{attribute 'enable_dynamic_creation'}
FUNCTION_BLOCK LineList EXTENDS CNM_AbstractObject.Object IMPLEMENTS ILineList
VAR
	list : CNM_Collections.ArrayList(1000);
END_VAR

(*

short summary
=================
This methode adds the given CNM_AbstractObject.IObject to the end of the list.
Example: 
Given a list that looks like this: (Head->) A B C (<- End),
calling append(D) on this list will place the D at the and,
making it the new End: (Head->) A B C D(<- End)

.. <legal notes>

legal notes
=================
| SPDX-FileCopyrightText: © 2022 ekvip automation GmbH <info@ekvip.de>
| SPDX-License-Identifier: Apache-2.0
| For details check: Apache-2.0_

.. _Apache-2.0: https://www.apache.org/licenses/LICENSE-2.0

.. </legal notes>

parameters
=================

*)
METHOD append : CNM_ReturnTypes.SingleExecutionResult
VAR_INPUT
	(*The object to be appended*)
	line	: ILine;
END_VAR
append := THIS^.list.append(object := line);
END_METHOD

(*

short summary
=================
This methode adds all elements of the given collection to the end of this list.
Example:
For the list1: A B C and list2: D E F will be after list1.appendCollection(list2):
A B C D E F. Notice the elements are still in the same order they where befor on each subsection.

.. <legal notes>

legal notes
=================
| SPDX-FileCopyrightText: © 2022 ekvip automation GmbH <info@ekvip.de>
| SPDX-License-Identifier: Apache-2.0
| For details check: Apache-2.0_

.. _Apache-2.0: https://www.apache.org/licenses/LICENSE-2.0

.. </legal notes>

parameters
=================

*)
METHOD appendCollection : CNM_ReturnTypes.SingleExecutionResult
VAR_INPUT
	(*The collection to be appended*)
	collectionToAppend	: CNM_CollectionInterfaces.ICollection;
END_VAR
appendCollection := THIS^.list.appendCollection(collectionToAppend);
END_METHOD

PROPERTY className : ClassName
GET
className := 'LineList';
END_GET
END_PROPERTY

(*

short summary
=================
This methode clears/deletes all clearable data from this object.
Example:
A list: 1 2 3 after list.clear() will have no remaining items, isEmpty = true.

.. <legal notes>

legal notes
=================
| SPDX-FileCopyrightText: © 2022 ekvip automation GmbH <info@ekvip.de>
| SPDX-License-Identifier: Apache-2.0
| For details check: Apache-2.0_

.. _Apache-2.0: https://www.apache.org/licenses/LICENSE-2.0

.. </legal notes>

parameters
=================

*)
METHOD clear
THIS^.list.clear();
END_METHOD

(*

short summary
=================
This methode checks if a given object is contained in the collection. 
The object is inside if the collection contains an object where the default comperator of the objects returns EQUAL on compareTo!

.. <legal notes>

legal notes
=================
| SPDX-FileCopyrightText: © 2022 ekvip automation GmbH <info@ekvip.de>
| SPDX-License-Identifier: Apache-2.0
| For details check: Apache-2.0_

.. _Apache-2.0: https://www.apache.org/licenses/LICENSE-2.0

.. </legal notes>

parameters
=================
:return: ``FALSE``: list does not contain an equal object
    ``TRUE``: list does contain an equal object

*)
METHOD containsEqualLine : BOOL
VAR_INPUT
	(*the object to be checked if it exists inside the collection*)
	line	: ILine;
END_VAR
containsEqualLine := THIS^.list.containsEqualObject(object := line);
END_METHOD

(*

short summary
=================
This methode checks if a given object is contained in the collection. 
The object is inside if the collection contains an object of equal hashcode!

.. <legal notes>

legal notes
=================
| SPDX-FileCopyrightText: © 2022 ekvip automation GmbH <info@ekvip.de>
| SPDX-License-Identifier: Apache-2.0
| For details check: Apache-2.0_

.. _Apache-2.0: https://www.apache.org/licenses/LICENSE-2.0

.. </legal notes>

parameters
=================
:return: ``FALSE``: list does not contain given object,
    ``TRUE``: list does contain given object

*)
METHOD containsLine : BOOL
VAR_INPUT
	(*the object to be checked if it exists inside the collection*)
	line	: ILine;
END_VAR
containsLine := THIS^.list.containsObject(object := line);
END_METHOD

{warning 'Add method implementation '}
(*

short summary
=================
This method is a self-destruction if the object was created dynamically.
If the object is a container class, the container content is destroyed with it.
The output NULL is a constant which is always NULL,
this allows a semi-pleasant notation: ``foo.deepDestruct(NULL => foo);``.

.. <legal notes>

legal notes
=================
| SPDX-FileCopyrightText: © 2022 ekvip automation GmbH <info@ekvip.de>
| SPDX-License-Identifier: Apache-2.0
| For details check: Apache-2.0_

.. _Apache-2.0: https://www.apache.org/licenses/LICENSE-2.0

.. </legal notes>

parameters
=================

InOut:
	+-----------------+------+---------+------------------------------------------+
	| Scope           | Name | Type    | Comment                                  |
	+=================+======+=========+==========================================+
	| Output CONSTANT | NULL | __XWORD | ``NULL`` is a constant which is always 0 |
	+-----------------+------+---------+------------------------------------------+

*)
METHOD deepDestruct
VAR_OUTPUT CONSTANT
	(* NULL is a constant which is always 0 *)
	NULL	: __XWORD;
END_VAR
THIS^.list.deepDestruct();
END_METHOD

(*

short summary
=================
This property returns the last object in the first and removes it from the list. Can be seen as opposite of prepend.
Example:
On a list: (Head -->) A B C, list.dequeue will return A.
Example 2:
If you call prepend(x), a dequeue right after will return x.

.. <legal notes>

legal notes
=================
| SPDX-FileCopyrightText: © 2022 ekvip automation GmbH <info@ekvip.de>
| SPDX-License-Identifier: Apache-2.0
| For details check: Apache-2.0_

.. _Apache-2.0: https://www.apache.org/licenses/LICENSE-2.0

.. </legal notes>

*)
METHOD dequeue : ILine
__QUERYINTERFACE(THIS^.list.dequeue(), dequeue);
END_METHOD

(*FB_Exit must be implemented explicitly. If there is an implementation, then the
method is called before the controller removes the code of the function block instance
(implicit call). The return value is not evaluated.*)
METHOD FB_Exit : BOOL
VAR_INPUT
	(* TRUE: the exit method is called in order to leave the instance which will be copied afterwards (online change).  *)
	bInCopyCode	: BOOL;
END_VAR
IF(THIS^.isObjectValid(THIS^.list))THEN
	THIS^.list.destruct();	
END_IF
END_METHOD

(*

short summary
=================
Method to perform a given action on all objects inside the collection.
Needs to reset the execution flag between calls.
Action to perform needs to implement :ref:`IApplier`.
Example:
You have a list of numbers: 1 2 3 and a ConcreteIncrementApplier that can take  a number and increment it. 
Calling list.forEach(TRUE, ConcreteIncrementApplier) will increment all numbers in the list, becoming: 2 3 4.

.. <legal notes>

legal notes
=================
| SPDX-FileCopyrightText: © 2022 ekvip automation GmbH <info@ekvip.de>
| SPDX-License-Identifier: Apache-2.0
| For details check: Apache-2.0_

.. _Apache-2.0: https://www.apache.org/licenses/LICENSE-2.0

.. </legal notes>

parameters
=========================
:return: CNM_ReturnTypes.ExecutionState

*)
METHOD forEach : CNM_ReturnTypes.SingleExecutionState
VAR_INPUT
	(*control bit to start or abort the forEach loop*)
	execute	: BOOL;
	(*the applier (action) to be used on all obejcts in the collection*)
	applier	: CNM_CollectionInterfaces.IApplier;
END_VAR
forEach := THIS^.list.forEach.parallel(execute := execute, applier := applier);
END_METHOD

(*

short summary
=================
This methode returns ths index of the first object that is equal to the given.
Example:
A list of: 1 2 3 after list.getIndexOf(1) will return: index=>0 and return IndexBounds.IN_BOUNDS
Example 2:
A list of: 1 2 3 after list.getIndexOf(4) will return: index=>3 and return IndexBounds.OUT_OF_BOUNDS

.. <legal notes>

legal notes
=================
| SPDX-FileCopyrightText: © 2022 ekvip automation GmbH <info@ekvip.de>
| SPDX-License-Identifier: Apache-2.0
| For details check: Apache-2.0_

.. _Apache-2.0: https://www.apache.org/licenses/LICENSE-2.0

.. </legal notes>

parameters
=================
:return: ``SingleExecutionResult.SUCCESS``: object found
    ``SingleExecutionResult.ERROR``: object couldn't be found in the list, index is undefined

*)
METHOD getIndexOf : CNM_ReturnTypes.SingleExecutionResult
VAR_INPUT
	(*the object to get the index from*)
	line	: ILine;
END_VAR
VAR_OUTPUT
	(*the index of the object inside the collection*)
	index	: __XWORD;
END_VAR
getIndexOf := THIS^.list.getIndexOf(object := line, index => index);
END_METHOD

(*

short summary
=================
This methode returns the object at the given index.
Returned objects can be modified, but not replaced! To replace an object use replaceObjectAt.
Example:
A list of: 1 2 3 after list.getObjectAt(1) will return: object=>2 and return SingleExecutionResult.SUCCESS
Example 2:
A list of: 1 2 3 after list.getObjectAt(3) will return: object=>NULL and return SingleExecutionResult.ERROR

.. <legal notes>

legal notes
=================
| SPDX-FileCopyrightText: © 2022 ekvip automation GmbH <info@ekvip.de>
| SPDX-License-Identifier: Apache-2.0
| For details check: Apache-2.0_

.. _Apache-2.0: https://www.apache.org/licenses/LICENSE-2.0

.. </legal notes>

parameters
=================
:return: ``SingleExecutionResult.SUCCESS``: index was valid
    ``SingleExecutionResult.ERROR``: index was not valid, returned object is undefined

*)
METHOD getLineAt : CNM_ReturnTypes.SingleExecutionResult
VAR_INPUT
	(*the index to access the object from*)
	index	: __XWORD;
END_VAR
VAR_OUTPUT
	(*the object at the given index*)
	line	: ILine;
END_VAR
VAR
	tmp : IObject;
END_VAR
getLineAt := THIS^.list.getObjectAt(index := index, object => tmp);
__QUERYINTERFACE(tmp, line);
END_METHOD

(*

short summary
=================
This property returns ``TRUE`` if the collection has any element.

.. <legal notes>

legal notes
=================
| SPDX-FileCopyrightText: © 2022 ekvip automation GmbH <info@ekvip.de>
| SPDX-License-Identifier: Apache-2.0
| For details check: Apache-2.0_

.. _Apache-2.0: https://www.apache.org/licenses/LICENSE-2.0

.. </legal notes>

*)
PROPERTY hasElement : BOOL
GET
hasElement := this^.list.hasElement;
END_GET
END_PROPERTY

(*

short summary
=================
This methode adds the given object at the given index. 
Will shift the other data starting at given index to the right.
List Lenght will be incremented.
Example:
A list of: 1 2 3 after list.insertObjectAt(1, object:=4) will become: 1 4 2 3 and return SingleExecutionResult.SUCCESS
Example 2:
A list of: 1 2 3 after list.insertObjectAt(3, object:=4) will become: 1 2 3 4 and return SingleExecutionResult.SUCCESS
Example 3:
A list of: 1 2 3 after list.insertObjectAt(5, object:=4) will become: 1 2 3 and return SingleExecutionResult.ERROR

.. <legal notes>

legal notes
=================
| SPDX-FileCopyrightText: © 2022 ekvip automation GmbH <info@ekvip.de>
| SPDX-License-Identifier: Apache-2.0
| For details check: Apache-2.0_

.. _Apache-2.0: https://www.apache.org/licenses/LICENSE-2.0

.. </legal notes>

parameters
=================
:return: ``SingleExecutionResult.SUCCESS``: index was valid, object inserted
    ``SingleExecutionResult.ERROR``: index out of bounds, list not changed

*)
METHOD insertLineAt : CNM_ReturnTypes.SingleExecutionResult
VAR_INPUT
	(*the index to insert the object at*)
	index	: __XWORD;
	(*the object to be added*)
	line	: ILine;
END_VAR
insertLineAt := THIS^.list.insertObjectAt(index := index, object := line);
END_METHOD

(*

short summary
=================
This method sorts the Sortable in the inverted order, so from great to low
.. <legal notes>

legal notes
=================
| SPDX-FileCopyrightText: © 2022 ekvip automation GmbH <info@ekvip.de>
| SPDX-License-Identifier: Apache-2.0
| For details check: Apache-2.0_

.. _Apache-2.0: https://www.apache.org/licenses/LICENSE-2.0

.. </legal notes>

parameters
=========================
:return: ``ABORTED``: While inverse was pending,execute had a falling edge,
	``BUSY``: Inverse is in progress
	``ERROR``: Inverse was not able to finish (p.e. List changed) call inverse(false) to reset
	``IDLE``: Currently invert is not in progress
	``SUCCESS``: Inversing was finished 
*)
METHOD inverseSort : CNM_ReturnTypes.SingleExecutionState
VAR_INPUT
	(*control bit to start or abort the inverting, needs to be active until the ExecutionState is noz longer busy*)
	execute	: BOOL;
END_VAR
inverseSort := THIS^.list.inverseSort(execute := execute);
END_METHOD

(*

short summary
=================
Inverts the order of the elements inside the object. Does not apply any kind of sorting, only reverses.

.. <legal notes>

legal notes
=================
| SPDX-FileCopyrightText: © 2022 ekvip automation GmbH <info@ekvip.de>
| SPDX-License-Identifier: Apache-2.0
| For details check: Apache-2.0_

.. _Apache-2.0: https://www.apache.org/licenses/LICENSE-2.0

.. </legal notes>

parameters
=========================

*)
METHOD invert
THIS^.list.invert();
END_METHOD

(*

short summary
=================
This property returns ``TRUE`` if the collection is empty.

.. <legal notes>

legal notes
=================
| SPDX-FileCopyrightText: © 2022 ekvip automation GmbH <info@ekvip.de>
| SPDX-License-Identifier: Apache-2.0
| For details check: Apache-2.0_

.. _Apache-2.0: https://www.apache.org/licenses/LICENSE-2.0

.. </legal notes>

*)
PROPERTY isEmpty : BOOL
GET
isEmpty := THIS^.list.isEmpty;
END_GET
END_PROPERTY

(*

short summary
=================
This methode returns the next object in the iteration and returns an execution state.
Example:
You have a list: 1 2 3
the first iterate call will return CNM_ReturnTypes.BUSY and object = 1
the second iterate call will return CNM_ReturnTypes.BUSY and object = 2
the third iterate call will return CNM_ReturnTypes.SUCCESS and object = 3

.. <legal notes>

legal notes
=================
| SPDX-FileCopyrightText: © 2022 ekvip automation GmbH <info@ekvip.de>
| SPDX-License-Identifier: Apache-2.0
| For details check: Apache-2.0_

.. _Apache-2.0: https://www.apache.org/licenses/LICENSE-2.0

.. </legal notes>

parameters
=================

*)
METHOD iterate : CNM_ReturnTypes.SingleExecutionState
VAR_INPUT
	(*control bit to start or abort the iterate*)
	execute	: BOOL;
END_VAR
VAR_OUTPUT
	(*the returned object of the iteration*)
	line	: ILine;
END_VAR
VAR
	tmp : IObject;
END_VAR
iterate := THIS^.list.iterate(execute := execute, object => tmp);
__QUERYINTERFACE(tmp, line);
END_METHOD

(*

short summary
=================
This property returns the last object in the list and removes it from the list. Can be seen as opposite of append.
Example:
On a list: (Head -->) A B C, list.pop will return C.
Example 2:
If you call append(x), a pop right after will return x.
May return a null pointer if list is empty

.. <legal notes>

legal notes
=================
| SPDX-FileCopyrightText: © 2022 ekvip automation GmbH <info@ekvip.de>
| SPDX-License-Identifier: Apache-2.0
| For details check: Apache-2.0_

.. _Apache-2.0: https://www.apache.org/licenses/LICENSE-2.0

.. </legal notes>

*)
METHOD pop : ILine
__QUERYINTERFACE(THIS^.list.pop(), pop);
END_METHOD

(*

short summary
=================
This methode adds the given obejct to the end of the list.
Example: 
Given a list that looks like this: (Head->) A B C (<- End),
calling prepend(D) on this list will place the D at start,
making it the new Head: (Head->) D A B C (<- End)

.. <legal notes>

legal notes
=================
| SPDX-FileCopyrightText: © 2022 ekvip automation GmbH <info@ekvip.de>
| SPDX-License-Identifier: Apache-2.0
| For details check: Apache-2.0_

.. _Apache-2.0: https://www.apache.org/licenses/LICENSE-2.0

.. </legal notes>

parameters
=================
:return: ``SingleExecutionResult.SUCCESS``: prepend was successful
	``SingleExecutionResult.ERROR``: allocation of memory for new object failed
	
*)
METHOD prepend : CNM_ReturnTypes.SingleExecutionResult
VAR_INPUT
	(*The object to be prepended*)
	line	: ILine;
END_VAR
prepend := THIS^.list.prepend(object := line);
END_METHOD

(*

short summary
=================
This methode adds all elements of the given collection to the start of this list. 
Example:
For the list1: A B C and list2: D E F will be after list1.prependCollection(list2):
D E F A B C. Notice the elements are still in the same order they where befor on each subsection.

.. <legal notes>

legal notes
=================
| SPDX-FileCopyrightText: © 2022 ekvip automation GmbH <info@ekvip.de>
| SPDX-License-Identifier: Apache-2.0
| For details check: Apache-2.0_

.. _Apache-2.0: https://www.apache.org/licenses/LICENSE-2.0

.. </legal notes>

parameters
=================
:return: ``SingleExecutionResult.SUCCESS``: prependCollection was successful
	``SingleExecutionResult.ERROR``: could not allocate memory for all new elements, list is left unchanged

*)
METHOD prependCollection : CNM_ReturnTypes.SingleExecutionResult
VAR_INPUT
	(*The collection to be prepended*)
	collectionToPrepend	: CNM_CollectionInterfaces.ICollection;
END_VAR
prependCollection := THIS^.list.prependCollection(collectionToPrepend := collectionToPrepend);
END_METHOD

(*

short summary
=================
This methode removes the first instance of the given object from the list.
Compares objects with hash value.
For example a Linked List: A B C A A D will on remove(A) becomes: B C A A D

.. <legal notes>

legal notes
=================
| SPDX-FileCopyrightText: © 2022 ekvip automation GmbH <info@ekvip.de>
| SPDX-License-Identifier: Apache-2.0
| For details check: Apache-2.0_

.. _Apache-2.0: https://www.apache.org/licenses/LICENSE-2.0

.. </legal notes>

parameters
=================

*)
METHOD remove
VAR_INPUT
	(*The object to be removed from the list*)
	line	: ILine;
END_VAR
THIS^.list.remove(object := line);
END_METHOD

(*

short summary
=================
This methode removes the element at the given index. 
Will shift the remaining data to the left (no empty space in list)
List Length will be decremented.
Example:
A list of: 1 2 3 after list.removeObjectAt(1) will become: 1 3 and return IndexBounds.IN_BOUNDS
Example 2:
A list of: 1 2 3 after list.removeObjectAt(3) will reamin: 1 2 3 and return IndexBounds.OUT_OF_BOUNDS

.. <legal notes>

legal notes
=================
| SPDX-FileCopyrightText: © 2022 ekvip automation GmbH <info@ekvip.de>
| SPDX-License-Identifier: Apache-2.0
| For details check: Apache-2.0_

.. _Apache-2.0: https://www.apache.org/licenses/LICENSE-2.0

.. </legal notes>

parameters
=================
:return: ``SingleExecutionResult.SUCCESS``: Element removed from index
    ``SingleExecutionResult.ERROR``: index out of bound, no object removed

*)
METHOD removeLineAt : CNM_ReturnTypes.SingleExecutionResult
VAR_INPUT
	(*the index to remove the object from*)
	index	: __XWORD;
END_VAR
removeLineAt := THIS^.list.removeObjectAt(index := index);
END_METHOD

(*

short summary
=================
This methode replaces the Interface reference inside the collection at the given index with the given Interface.
Example:
A list of: 1 2 3 after list.replaceObjectAt(1, withObject:=4) will become: 1 4 3 and return SingleExecutionResult.SUCCESS
Example 2:
A list of: 1 2 3 after list.replaceObjectAt(3, withObject:=4) will remain: 1 2 3 and return SingleExecutionResult.ERROR

.. <legal notes>

legal notes
=================
| SPDX-FileCopyrightText: © 2022 ekvip automation GmbH <info@ekvip.de>
| SPDX-License-Identifier: Apache-2.0
| For details check: Apache-2.0_

.. _Apache-2.0: https://www.apache.org/licenses/LICENSE-2.0

.. </legal notes>

parameters
=================
:return: ``SingleExecutionResult.SUCCESS``: index valid, element at index replaced with ``withObject``
    ``SingleExecutionResult.ERROR``: ìndex out of bounds, nothing changed

*)
METHOD replaceLineAt : CNM_ReturnTypes.SingleExecutionResult
VAR_INPUT
	(*the index to replace the object at*)
	index	: __XWORD;
	(*the object to be at this index instead*)
	withLine	: ILine;
END_VAR
replaceLineAt := THIS^.list.replaceObjectAt(index := index, withObject := withLine);
END_METHOD

(*

short summary
=================
This methode can replace the default sorter for a custom one. Check :ref:`IListSorter`
Can be used for performant sorting algorithms if more about the data structure is known.

.. attention:: 
	For implementations: **IListSorter is an empty interface and you should extend it with custom interfaces for each type of list.**
	For LinkedList see :ref:`ILinkedListSorter`. 
	Your implementation should then use this extended interface and the setter should check for compability. 
	
.. <legal notes>

legal notes
=================
| SPDX-FileCopyrightText: © 2022 ekvip automation GmbH <info@ekvip.de>
| SPDX-License-Identifier: Apache-2.0
| For details check: Apache-2.0_

.. _Apache-2.0: https://www.apache.org/licenses/LICENSE-2.0

.. </legal notes>

parameters
=================
:return: ``THIS^`` :ref:`IList`

*)
METHOD setSorter : CNM_CollectionInterfaces.ISortable
VAR_INPUT
	(*The instance of the sorter to be used to sort the list*)
	sorter	: CNM_CollectionInterfaces.IArrayListSorter;
END_VAR
setSorter := THIS^.list.setSorter(sorter := sorter);
END_METHOD

(*

short summary
=================
This property returns the number of elements inside this collection.

.. <legal notes>

legal notes
=================
| SPDX-FileCopyrightText: © 2022 ekvip automation GmbH <info@ekvip.de>
| SPDX-License-Identifier: Apache-2.0
| For details check: Apache-2.0_

.. _Apache-2.0: https://www.apache.org/licenses/LICENSE-2.0

.. </legal notes>

*)
PROPERTY size : __XWORD
GET
size := THIS^.list.size;
END_GET
END_PROPERTY

(*

short summary
=================
This method sorts the data structure. 
This can take many cycles and should be called until the CNM_ReturnTypes.ExecutionState is no longer ``BUSY``.

.. <legal notes>

legal notes
=================
| SPDX-FileCopyrightText: © 2022 ekvip automation GmbH <info@ekvip.de>
| SPDX-License-Identifier: Apache-2.0
| For details check: Apache-2.0_

.. _Apache-2.0: https://www.apache.org/licenses/LICENSE-2.0

.. </legal notes>

parameters
=================
:return: ``ABORTED``: While sort was pending,execute had a falling edge,
	``BUSY``: Sort is in progress
	``ERROR``: Sort was not able to finish (p.e. List changed) call sort(false) to reset
	``IDLE``: Currently no sort in progress
	``SUCCESS``: Sorting was finished 

*)
METHOD sort : CNM_ReturnTypes.SingleExecutionState
VAR_INPUT
	(*control bit to start or abort the sorting, needs to be active until the ExecutionState is SUCCESS*)
	execute	: BOOL;
END_VAR
sort := THIS^.list.sort(execute := execute);
END_METHOD

(*

short summary
=================
This method sorts the data structure. 
It uses the passed Comperator to sort the structure.
This can take many cycles and should be called until the CNM_ReturnTypes.ExecutionState is no longer ``BUSY``.

.. <legal notes>

legal notes
=================
| SPDX-FileCopyrightText: © 2022 ekvip automation GmbH <info@ekvip.de>
| SPDX-License-Identifier: Apache-2.0
| For details check: Apache-2.0_

.. _Apache-2.0: https://www.apache.org/licenses/LICENSE-2.0

.. </legal notes>

parameters
=================
:return: ``ABORTED``: While sort was pending,execute had a falling edge,
	``BUSY``: Sort is in progress
	``ERROR``: Sort was not able to finish (p.e. List changed) call sort(false) to reset
	``IDLE``: Currently no sort in progress
	``SUCCESS``: Sorting was finished 

*)
METHOD sortWithComparator : CNM_ReturnTypes.SingleExecutionState
VAR_INPUT
	(*control bit to start or abort the sorting, needs to be active until the ExecutionState is SUCCESS*)
	execute	: BOOL;
	(*the comparator that should be used for the sort. Must not be changed while sort is in process*)
	comparator	: CNM_AbstractObject.IComparator;
END_VAR
sortWithComparator := THIS^.list.sortWithComparator(execute := execute, comparator := comparator);
END_METHOD

END_FUNCTION_BLOCK

(* stored: Version 1.1.0.1
   POU LineList: Id {b15030db-490d-4ef0-82d7-005c853e7ace}, SpecialFunc None
   Folder Object: Id {c1ed7c17-6094-4cb2-bdd0-4ac6ea061379}
   Method append: Id {13a53413-be7d-4921-a53c-36f48fa8332d}
   Method appendCollection: Id {fbbab5bd-a80f-4b62-a9f2-8e8341a1cf63}
   Property className: Id {09660b95-41e7-4768-8afe-6c8d001b2d58}
   Get Get: Id {4c4a5ba2-2160-48c3-82ae-2e0d96bbe826}
   Method clear: Id {c7c49bbe-4390-43ff-8441-796063364e99}
   Method containsEqualLine: Id {c2634b06-17ae-451d-b0dc-38eee6dbb592}
   Method containsLine: Id {2ca1f51a-5fae-4c58-a457-de1aa0e1b380}
   Method deepDestruct: Id {da945ed7-0d84-4082-b7c3-46116ee5cbf1}
   Method dequeue: Id {1d15acef-0c5f-42a3-8c2b-122571dbbf5e}
   Method FB_Exit: Id {bea76fb4-ab5b-46fa-8dc4-0a69dd1248a2}
   Method forEach: Id {a0abab77-e660-4b68-ba39-d74e2c5f560d}
   Method getIndexOf: Id {ec3cc899-95e7-476d-ad39-74296dd8ca64}
   Method getLineAt: Id {396b6100-38f1-4e33-8371-983075989e6d}
   Property hasElement: Id {22a015fd-b82d-40b8-bfc5-dd63c8a9e913}
   Get Get: Id {19d62138-6b0c-4097-8db3-a79d9e233566}
   Method insertLineAt: Id {2fbf4c99-7123-4a13-b1c3-7c351e9c4324}
   Method inverseSort: Id {6dcf984a-3c19-423b-b73c-6c6fd8a0853f}
   Method invert: Id {9dbb1161-c660-488d-91e4-2ea9b99c5778}
   Property isEmpty: Id {27fae613-0223-4dda-afa2-aafe28368d05}
   Get Get: Id {db0f414e-933a-4e46-a50b-54262846d171}
   Method iterate: Id {93ffdfe0-3bdf-46ee-aeb7-6b3a37d476a0}
   Method pop: Id {4f16b8a1-8f09-4946-85c0-18b8451b469a}
   Method prepend: Id {a29599cd-ea2a-45c5-9cd5-6808ca9e13d5}
   Method prependCollection: Id {b5c5b302-ca05-493f-aab6-a0ef8ae307fc}
   Method remove: Id {56668ef7-6583-4672-bf47-952e7b8805f5}
   Method removeLineAt: Id {121d0344-1d7b-4260-b99a-adc951aa8da4}
   Method replaceLineAt: Id {37f4d5cb-7445-4bf8-9053-ca090cac4009}
   Method setSorter: Id {3e5c7620-4a37-44cf-8f4c-a72506d7ae62}
   Property size: Id {9b80adba-7a6f-40c8-989d-c322552f0e2c}
   Get Get: Id {3ac1a34d-e753-4766-af5a-4364c6721699}
   Method sort: Id {23a5b5f9-e8ac-4d52-9729-dd962b98cb5e}
   Method sortWithComparator: Id {1db1b1f5-d2d8-47be-9b50-a61e9d327c8e} *)
